PROGRAM MAIN
VAR
	bLED1	AT%Q* : BOOL;
END_VAR

bLED1 := TRUE;

END_PROGRAM

(* stored: Version 1.1.0.1, ProductVersion 3.1.4022.3
   POU MAIN: Id {f58e1d9e-fe57-40b8-989d-e2e4f67a8ce2}, SpecialFunc None *)
